TYPE
    TcaLaserDistanceSenorConfig :
    STRUCT
        RawLow   : DINT;
        RawHigh  : DINT;
        RealLow  : REAL;
        RealHigh : REAL;
        Gain     : REAL := 1.0;
        Offset   : REAL := 0.0;
    END_STRUCT
END_TYPE

(* stored: Version 1.1.0.1
   DUT TcaLaserDistanceSenorConfig: Id {31493de9-7001-4ccb-b01f-48bd508f2dfd} *)
